Universal Robots PolyScope program: Put_into_box_UR10.urp

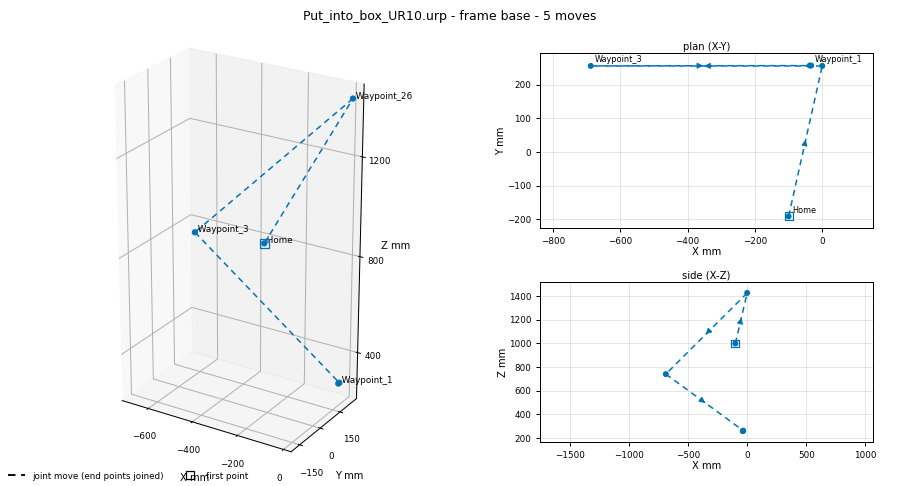
[picture p0: tool path of Put_into_box_UR10.urp in frame base, 5 of 5 moves have a stored position in this frame; points joined in program order, loops and branches not executed]
ProgramRoot directory=/home/ur/ursim-1.5/programs/templates/PutIntoBox; kinematics=(a=[0, -0.425, -0.39243, 0, 0, 0], d=[0.0892, 0, 0, 0.109, 0.093, 0.082], alpha=[1.5708, 0, 0, 1.5708, -1.5708, 0], deltaTheta=[0, 0, 0, 0, 0, 0], status=notInitialized); name=Put_into_box_UR10; programVersion=(project__name=PolyScope, major__version=1, minor__version=0, svn__revision=0); robotEnvironmentFileName=default; variables=(Variable=(name=loop_1, prefersPersistentValue=false, requestANewUniqueName=false), Variable=(name=loop_2, prefersPersistentValue=false, requestANewUniqueName=false), Variable=(name=loop_3, prefersPersistentValue=false, requestANewUniqueName=false), Variable=(name=loop_4, prefersPersistentValue=false, requestANewUniqueName=false), Variable=(name=loop_5, prefersPersistentValue=false, requestANewUniqueName=false), Variable=(name=loop_6, prefersPersistentValue=false, requestANewUniqueName=false), Variable=(name=loop_7, prefersPersistentValue=false, requestANewUniqueName=false))
  MainProgram cartesianAcceleration=1.2; cartesianSpeed=0.3; jointAcceleration=1.3962634015954636; jointSpeed=1.0471975511965976; moveAsFastAsPossible=true; sharedProcessMoveBlendRadius=0.0; featureReference=(installationNameReference=Base); motionType=JOINT_SPACE; runOnlyOneCycle=true
    Action analogValue=4.0; digitalValue=0; payloadValue=0.0; selectedAnalogSensor=-1; selectedDigitalSensor=-1; setPayloadValue=true; type=NO_ACTION
    Move cartesianAcceleration=1.2; cartesianSpeed=0.3; jointAcceleration=1.7453292519943295; jointSpeed=0.8726646259971648; moveAsFastAsPossible=true; sharedProcessMoveBlendRadius=0.025; featureReference=(installationNameReference=Base); motionType=JOINT_SPACE
      Waypoint blendRadius=0.0; cartesianAcceleration=1.2; cartesianSpeed=0.3; jointAcceleration=1.3962634015954636; jointSpeed=1.0471975511965976; nextMotionTime=2.0; stoppoint=true; useSharedParameters=true; position=TCP in base x=-99.993 y=-190.994 z=999.647 mm, rx=0.0001 ry=-2.2213 rz=2.2213 rad; joints [0, -90, 0, -90, 0, 0] deg; positionType=FIXED_POSITION; name=Home
      Popup message=Remove the 2 screws in base pointing towards the cable attachment; type=MESSAGE
      Waypoint blendRadius=0.05; cartesianAcceleration=1.2; cartesianSpeed=0.3; jointAcceleration=1.3962634015954636; jointSpeed=1.0471975511965976; nextMotionTime=2.0; stoppoint=true; useSharedParameters=true; position=TCP in base x=0 y=256.141 z=1427.3 mm, rx=-1.5708 ry=0 rz=0 rad; joints [-180, -90, 0, -90, 0, 0] deg; positionType=FIXED_POSITION; waypointPoseInFeatureCoordinates=(pos=(x=-5.655634450898706E-16, y=0.256141000242904, z=1.4272999999474645), rot=(x=-1.570796327, y=-9.562469296879588E-16, z=1.2997498003256397E-15)); name=Waypoint_26
      Waypoint blendRadius=0.05; cartesianAcceleration=1.2; cartesianSpeed=0.25; jointAcceleration=1.3962634015954636; jointSpeed=1.0471975511965976; nextMotionTime=2.0; stoppoint=true; useSharedBlendParameter=true; useSharedParameters=true; position=TCP in base x=-687.999 y=256.141 z=740.645 mm, rx=-1.2101 ry=-1.2078 rz=-1.2078 rad; joints [-180, -90, -89.888, -90, 0, 0] deg; positionType=FIXED_POSITION; waypointPoseInFeatureCoordinates=(pos=(x=-0.6879986847842301, y=0.25614100010206775, z=0.7406452639251114), rot=(x=-1.2101234171267714, y=-1.2077595407064616, z=-1.2077595404587445)); name=Waypoint_3
      Popup message=Check for any external wiring etc. to prevent any damage; type=MESSAGE
      Waypoint blendRadius=0.05; cartesianAcceleration=1.2; cartesianSpeed=0.25; jointAcceleration=1.3962634015954636; jointSpeed=1.0471975511965976; nextMotionTime=2.0; stoppoint=true; useSharedBlendParameter=true; useSharedParameters=true; position=TCP in base x=-32.878 y=257.156 z=262.435 mm, rx=-1.2554 ry=-1.1877 rz=-1.201 rad; joints [-181.616, 6.179, -164.784, -109.841, 0.996, 0.033] deg; positionType=FIXED_POSITION; waypointPoseInFeatureCoordinates=(pos=(x=-0.032878049003463326, y=0.25715646817308513, z=0.26243500342076703), rot=(x=-1.2553807735860671, y=-1.187658989189511, z=-1.2009606962629082)); name=Waypoint_1
      Popup message=Place protective pad between arm and base joint; type=MESSAGE
      Waypoint blendRadius=0.05; cartesianAcceleration=1.2; cartesianSpeed=0.25; jointAcceleration=1.3962634015954636; jointSpeed=1.0471975511965976; nextMotionTime=2.0; stoppoint=true; useSharedBlendParameter=true; useSharedParameters=true; position=TCP in base x=-37.267 y=257.28 z=257.678 mm, rx=-1.2457 ry=-1.2038 rz=-1.217 rad; joints [-181.616, 6.179, -166.022, -109.841, 0.996, 0.033] deg; positionType=FIXED_POSITION; waypointPoseInFeatureCoordinates=(pos=(x=-0.037267417312010824, y=0.2572802936718336, z=0.25767812473840873), rot=(x=-1.245693230202273, y=-1.2038044945179394, z=-1.2169975619132969)); name=Waypoint_2
